FUNCTION_BLOCK escalonamento (* Composite Function Block Type *)
  (* Standard: 61499-2 *)
  (* Version 0.0, 1/29/2026, Schneider Electric, template *)
  PACKAGE Hidryco.HidrycoLib;
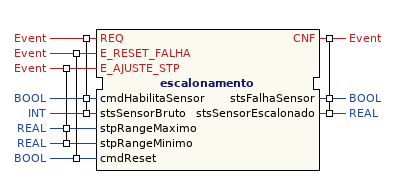
  EVENT_INPUT
    REQ WITH cmdHabilitaSensor, stsSensorBruto; (* Normal Execution Request *)
    E_RESET_FALHA WITH cmdReset;
    E_AJUSTE_STP WITH stpRangeMaximo, stpRangeMinimo;
  END_EVENT
  EVENT_OUTPUT
    CNF WITH stsFalhaSensor, stsSensorEscalonado; (* Execution Confirmation *)
  END_EVENT
  VAR_INPUT
    cmdHabilitaSensor : BOOL;
    stsSensorBruto : INT; (* Input event qualifier *)
    stpRangeMaximo : REAL;
    stpRangeMinimo : REAL;
    cmdReset : BOOL;
  END_VAR
  VAR_OUTPUT
    stsFalhaSensor : BOOL;
    stsSensorEscalonado : REAL;
  END_VAR
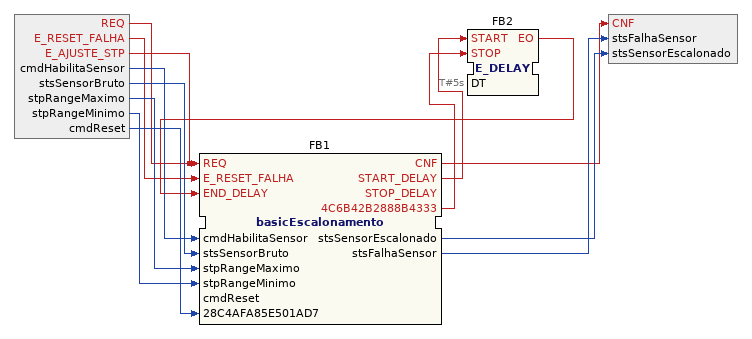
  FBS
    FB1 : basicEscalonamento;
    FB2 : E_DELAY(DT := T#5s);
  END_FBS
  EVENT_CONNECTIONS
    E_RESET_FALHA TO FB1.E_RESET_FALHA;
    REQ TO FB1.REQ;
    FB1.CNF TO CNF;
    FB1.START_DELAY TO FB2.START;
    FB2.EO TO FB1.END_DELAY;
    FB1.4C6B42B2888B4333 TO FB2.STOP;
    E_AJUSTE_STP TO FB1.REQ;
  END_CONNECTIONS
  DATA_CONNECTIONS
    stpRangeMinimo TO FB1.stpRangeMinimo;
    stpRangeMaximo TO FB1.stpRangeMaximo;
    stsSensorBruto TO FB1.stsSensorBruto;
    cmdHabilitaSensor TO FB1.cmdHabilitaSensor;
    FB1.stsSensorEscalonado TO stsSensorEscalonado;
    FB1.stsFalhaSensor TO stsFalhaSensor;
    cmdReset TO FB1.28C4AFA85E501AD7;
  END_CONNECTIONS
END_FUNCTION_BLOCK
